FUNCTION_BLOCK ROBOT6TESTFB (* JADE WORKER *)
  (* Standard: 61499-1 *)
  (* Version 1.0, 2014-04-22, Ahmed, Fraunhofer IGD *)
  (* Compiler header: package fb.rt; *)
  (* Compiler Java Sun JDK 1.5.0 *)
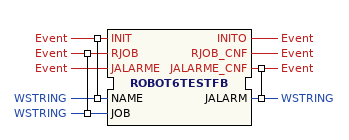
  EVENT_INPUT
    INIT WITH NAME; (* Normal Execution Request *)
    RJOB WITH JOB; (* Normal Execution Request *)
    JALARME;
  END_EVENT
  EVENT_OUTPUT
    INITO; (* Execution Confirmation *)
    RJOB_CNF; (* Execution Confirmation *)
    JALARME_CNF WITH JALARM;
  END_EVENT
  VAR_INPUT
    NAME : WSTRING;
    JOB : WSTRING;
  END_VAR
  VAR_OUTPUT
    JALARM : WSTRING;
  END_VAR
END_FUNCTION_BLOCK
